TYPE T_CoEIndex : WORD; END_TYPE

(* stored: Version 1.1.0.1, ProductVersion 3.1.4024.14
   DUT T_CoEIndex: Id {45e8fab0-1a6e-0024-0243-27b13133f2be} *)
